TYPE ST_Memory_Info :
STRUCT
	rTotal			: REAL;
	rUsage			: REAL;
	rUsage_percent	: REAL;
	sTotal			: STRING(20);
	sUsage			: STRING(20);	
END_STRUCT
END_TYPE

(* stored: Version 1.1.0.1, ProductVersion 3.1.4022.18
   DUT ST_Memory_Info: Id {fe219a10-6f0d-4ed0-842c-5c675fe8ed4e} *)
